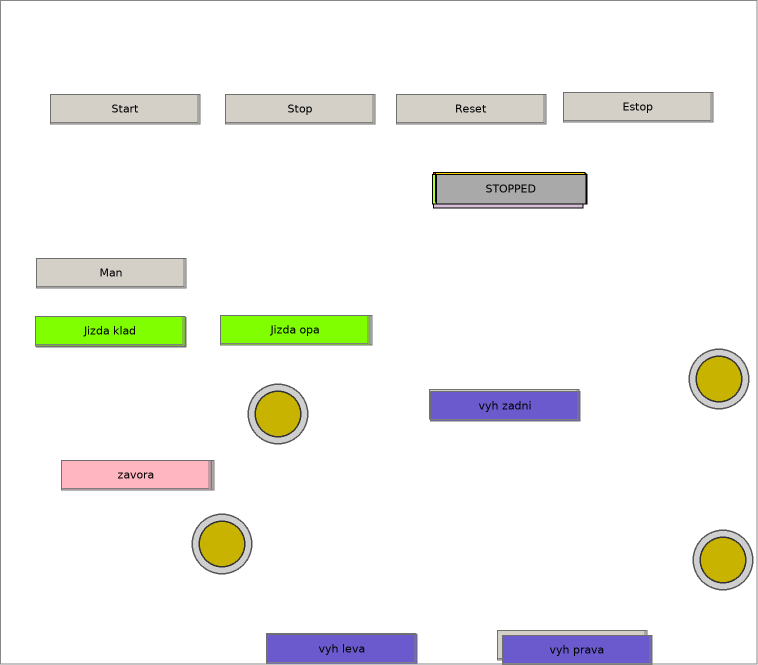
VISUALIZATION Visualization  // 758x665
    Button (50,94 150x30), "Start"
        tap SCADA.SCADA_START
    Button (225,94 150x30), "Stop"
        tap SCADA.SCADA_STOP
    Button (36,258 150x30), "Man", input disabled if: SCADA.systemstav=11
        tap SCADA.SCADA_MAN
    Button (396,94 150x30), "Reset"
        tap SCADA.SCADA_RESET
    Button (36,317 150x30), "Jizda klad", input disabled if: SCADA.systemstav<>11
        toggle SCADA.SCADA_MAN_OPACNY
    Button (64,460 150x30), "zavora", input disabled if: SCADA.systemstav<>11
        OnMouseClick: toggle SCADA.SCADA_MAN_ZAVORY
    Button (497,630 150x30), "vyh prava", input disabled if: SCADA.systemstav<>11
        tap SCADA.SCADA_MAN_IMP_PRA
    Button (429,389 150x30), "vyh zadni", input disabled if: SCADA.systemstav<>11
        tap SCADA.SCADA_MAN_IMP_ZAD
    Button (266,633 150x30), "vyh leva", input disabled if: SCADA.systemstav<>11
        tap SCADA.SCADA_MAN_IMP_LEV
    Button (222,315 150x30), "Jizda opa", input disabled if: SCADA.systemstav<>11
        toggle SCADA.SCADA_MAN_KLADNY
    Button (563,92 150x30), "Estop"
        toggle SCADA.SCADA_ESTOP
    Lamp1 (243,379 70x70), variable: TAGS.HRA_ZAV, style: Lamp-Lamp1-Yellow
    Lamp1 (187,509 70x70), variable: TAGS.HRA_LEV, style: Lamp-Lamp1-Yellow
    Lamp1 (688,525 70x70), variable: TAGS.HRA_PRA, style: Lamp-Lamp1-Yellow
    Lamp1 (684,344 70x70), variable: TAGS.HRA_ZAD, style: Lamp-Lamp1-Yellow
    Rectangle (436,173 150x30), "MANUAL", text variable: SCADA.systemstav, invisible if: SCADA.systemstav<>11
    Rectangle (433,178 150x30), "CLEARING", text variable: SCADA.systemstav, invisible if: SCADA.systemstav<>10
    Rectangle (433,172 150x30), "ABORTED", text variable: SCADA.systemstav, invisible if: SCADA.systemstav<>9
    Rectangle (435,173 150x30), "COMPLETE. Press Reset", text variable: SCADA.systemstav, invisible if: SCADA.systemstav<>7
    Rectangle (437,174 150x30), "HELD", text variable: SCADA.systemstav, invisible if: SCADA.systemstav<>4
    Rectangle (432,174 150x30), "Running", text variable: SCADA.systemstav, invisible if: SCADA.systemstav<>2
    Rectangle (435,172 150x30), "STARTING", text variable: SCADA.systemstav, invisible if: SCADA.systemstav<>1
    Rectangle (436,174 150x30), "STOPPED", text variable: SCADA.systemstav, invisible if: SCADA.systemstav<>0
    Button (35,316 150x30), "Jizda klad", invisible if: NOT MAIN.fbDrive.outKLADNY
        toggle SCADA.SCADA_MAN_OPACNY
    Button (220,315 150x30), "Jizda opa", invisible if: NOT MAIN.fbDrive.outOPACNY
        toggle SCADA.SCADA_MAN_KLADNY
    Button (61,460 150x30), "zavora", invisible if: NOT TAGS.ZAVORY, input disabled if: SCADA.systemstav<>11
        OnMouseClick: toggle SCADA.SCADA_MAN_ZAVORY
    Button (267,634 150x30), "vyh leva", invisible if: NOT TAGS.VYH_LEV, input disabled if: SCADA.systemstav<>11
        tap SCADA.SCADA_MAN_IMP_LEV
    Button (502,635 150x30), "vyh prava", invisible if: NOT TAGS.VYH_PRA, input disabled if: SCADA.systemstav<>11
        tap SCADA.SCADA_MAN_IMP_PRA
    Button (430,391 150x30), "vyh zadni", invisible if: NOT TAGS.VYH_ZAD, input disabled if: SCADA.systemstav<>11
        tap SCADA.SCADA_MAN_IMP_ZAD
END_VISUALIZATION

(* stored: Version 1.1.0.1, ProductVersion 3.1.4024.13
   Visu Visualization: Id {db30e378-f933-4933-9d39-e65678c40337} *)
